FUNCTION_BLOCK SAT IMPLEMENTS MachineModule
VAR
	bEnable			: BOOL;
	bDisable        : BOOL;
	bError          : BOOL;
	bOverride       : BOOL;
	bSimulation     : BOOL;
	bStart          : BOOL;
	bStop           : BOOL;
END_VAR

// This is the core module needed that we are creating for our STS and contains everything related to the STS

// To be added
(*
FEEDER

SAT

VBT

EJECT

GATE

SBT

*)

METHOD Disable : BOOL
VAR_INPUT
END_VAR
bEnable:=FALSE;
END_METHOD

METHOD Enable : BOOL
VAR_INPUT
END_VAR
bEnable:=TRUE;
bDisable:=False;
END_METHOD

METHOD Error : BOOL
VAR_INPUT
END_VAR
bEnable:=FALSE;
END_METHOD

METHOD Override : BOOL
VAR_INPUT
END_VAR
END_METHOD

METHOD Reset : BOOL
VAR_INPUT
END_VAR
END_METHOD

METHOD Start : BOOL
VAR_INPUT
END_VAR
END_METHOD

METHOD PUBLIC StateMachine
VAR_INPUT
END_VAR
END_METHOD

METHOD Stop : BOOL
VAR_INPUT
END_VAR
END_METHOD

END_FUNCTION_BLOCK

(* stored: Version 1.1.0.1, ProductVersion 3.1.4024.12
   POU SAT: Id {948e0ac6-ae65-4c94-b7cd-dfb2a0ed80d3}, SpecialFunc None
   Method Disable: Id {5e86057e-6890-4f43-bb81-e98513f8c202}
   Method Enable: Id {71274df4-0a05-4959-b444-38e8c80a464b}
   Method Error: Id {0ab8f348-744d-48b4-b5e0-eaebf6040d04}
   Method Override: Id {927c0db9-5b10-4b75-ba46-3e285b30c6ad}
   Method Reset: Id {b6d1550e-3880-446a-9451-6a93dd56d0bf}
   Method Start: Id {7a2b105a-6841-4d93-8a66-d106007db900}
   Method StateMachine: Id {c6dcb0ef-7831-4a12-af30-96f167333d50}
   Method Stop: Id {892d6684-3aec-4152-8a75-d7d9c0ca91de} *)
